(* IEC 61131-3 sources: teller/JD_Teller_LC2_V11/Class/TellerClass_Teller, 1 file *)

(* ---- TellerClass_Teller.st ---- *)
(*!
<Class
	Name               = "TellerClass_Teller"
	Revision           = "1.3"
	RealtimeTask       = "true"
	DefRealtime        = "1 ms"
	DefRealtimeIndex   = "1073742080"
	CyclicTask         = "true"
	DefCyclictime      = "100 ms"
	DefCyclicIndex     = "1073742080"
	BackgroundTask     = "true"
	DefBackground      = "200 ms"
	DefBackgroundIndex = "1073742080"
	Sigmatek           = "false"
	OSInterface        = "false"
	HighPriority       = "false"
	Automatic          = "false"
	UpdateMode         = "Prescan"
	SharedCommandTable = "true"
	Objectsize         = "(570,120)">
	<Channels>
		<Server Name="ClassSvr" Visualized="true" Initialize="false" WriteProtected="false" Retentive="false" Comment="Standaard 20&#13;&#10;"/>
		<Server Name="i2SenCNT" Visualized="true" Initialize="false" WriteProtected="false" Retentive="false" Comment="Servicemenu instelling&#13;&#10;&#13;&#10;Met de waarde kan het aantal telsensors worden ingesteld.&#13;&#10;Algemene instelling. Met deze server worden alle Visuteller &#13;&#10;i2SenCNT overschreven!&#13;&#10;&#13;&#10;Bereik&#13;&#10;&#13;&#10;0:&#13;&#10;Alleen SensorL wordt gebruikt bij type 1 t/m 5, behalve type 3.&#13;&#10;&#13;&#10;1:&#13;&#10;Zowel Sensor L en Sensor R worden gebruikt bij type 1t/m 5, behalve type 3.&#13;&#10;&#13;&#10;"/>
		<Server Name="iBoxlengthCNT" Visualized="true" Initialize="false" WriteProtected="false" Retentive="false"/>
		<Server Name="iBoxlengthCNT_Max" Visualized="true" Initialize="false" WriteProtected="true" Retentive="false"/>
		<Server Name="iBoxlengthCNT_Min" Visualized="true" Initialize="false" WriteProtected="true" Retentive="false"/>
		<Server Name="iBoxlengthJamL" Visualized="true" Initialize="false" WriteProtected="false" Retentive="false"/>
		<Server Name="iBoxlengthJamL_Max" Visualized="true" Initialize="false" WriteProtected="true" Retentive="false"/>
		<Server Name="iBoxlengthJamL_Min" Visualized="true" Initialize="false" WriteProtected="true" Retentive="false"/>
		<Server Name="iBoxlengthJamR" Visualized="true" Initialize="false" WriteProtected="false" Retentive="false"/>
		<Server Name="iBoxlengthJamR_Max" Visualized="true" Initialize="false" WriteProtected="true" Retentive="false"/>
		<Server Name="iBoxlengthJamR_Min" Visualized="true" Initialize="false" WriteProtected="true" Retentive="false"/>
		<Server Name="iBoxlengthJamSTR" Visualized="true" Initialize="false" WriteProtected="false" Retentive="false"/>
		<Server Name="iBoxlengthJamSTR_Max" Visualized="true" Initialize="false" WriteProtected="true" Retentive="false"/>
		<Server Name="iBoxlengthJamSTR_Min" Visualized="true" Initialize="false" WriteProtected="true" Retentive="false"/>
		<Server Name="iEncDiv" Visualized="true" Initialize="false" WriteProtected="false" Retentive="false" Comment="idem als iEncMul&#13;&#10;&#13;&#10;Alleen is dit de deelfactor"/>
		<Server Name="iEncMeetdist" Visualized="true" Initialize="false" WriteProtected="false" Retentive="false"/>
		<Server Name="iEncMul" Visualized="true" Initialize="false" WriteProtected="false" Retentive="false" Comment="Met deze instelling is de encoder in te stellen naar de juiste eenheid.&#13;&#10;&#13;&#10;Dit is de vermenigvuldig factor&#13;&#10;&#13;&#10; "/>
		<Server Name="iEncStapper" Visualized="true" Initialize="false" WriteProtected="false" Retentive="false"/>
		<Server Name="iJamdetReset" Visualized="true" Initialize="false" WriteProtected="false" Retentive="false"/>
		<Server Name="iSensorCNT" Visualized="true" Initialize="false" WriteProtected="false" Retentive="false" Comment="&#13;&#10;&#13;&#10;"/>
		<Server Name="iTotalProduction" Visualized="true" Initialize="false" WriteProtected="false" Retentive="false"/>
		<Server Name="MinSpot" Visualized="true" Initialize="false" WriteProtected="false" Retentive="false"/>
		<Server Name="oCounter" Visualized="true" Initialize="false" WriteProtected="false" Retentive="false"/>
		<Server Name="oCounterPerHour" Visualized="true" Initialize="false" WriteProtected="false" Retentive="false"/>
		<Server Name="oJamdetL" Visualized="true" Initialize="false" WriteProtected="true" Retentive="false"/>
		<Server Name="oJamdetR" Visualized="true" Initialize="false" WriteProtected="true" Retentive="false"/>
		<Server Name="oJamdetSTR" Visualized="true" Initialize="false" WriteProtected="true" Retentive="false"/>
		<Server Name="oRemainingProduction" Visualized="true" Initialize="false" WriteProtected="false" Retentive="false"/>
		<Server Name="oSensorHWCNT" Visualized="true" Initialize="false" WriteProtected="true" Retentive="false"/>
		<Server Name="oSpeed" Visualized="true" Initialize="false" WriteProtected="true" Retentive="false" Comment="Snelheid machine in m/min.&#13;&#10;&#13;&#10;in meter per minuut.&#13;&#10;"/>
		<Server Name="oStopperLSE" Visualized="true" Initialize="false" WriteProtected="false" Retentive="false" Comment="De serverLSE wordt gebruikt om plaatjes in LSE te laten zien"/>
		<Server Name="sAnalogSpeed_Man_Auto" Visualized="true" Initialize="false" WriteProtected="false" Retentive="false"/>
		<Server Name="sAnalogSpeedEnable" Visualized="true" Initialize="false" WriteProtected="false" Retentive="false"/>
		<Server Name="sCounter" Visualized="false" Initialize="false" WriteProtected="true" Retentive="false"/>
		<Server Name="sCounterPerMin" Visualized="false" Initialize="false" WriteProtected="true" Retentive="false"/>
		<Server Name="sData" Visualized="false" Initialize="false" WriteProtected="false" Retentive="SRam"/>
		<Server Name="SExtraBox" Visualized="true" Initialize="false" WriteProtected="false" Retentive="false" Comment="Standaard 30"/>
		<Server Name="sFactorAnalogSpeedIn" Visualized="true" Initialize="false" WriteProtected="false" Retentive="false" Comment="Slider voor bepaling van een factor voor aansturing van de conveyor met een analoog signaal&#13;&#10;&#13;&#10;Min = 0&#13;&#10;Max = 10000"/>
		<Server Name="sFactorAnalogSpeedout" Visualized="true" Initialize="false" WriteProtected="true" Retentive="false" Comment="&#13;&#10;Output voor snelheids referentie van de conveyor&#13;&#10;Factor voor aansturing van de conveyor met een analoog signaal&#13;&#10;&#13;&#10;Min = 0&#13;&#10;Max = 10000"/>
		<Server Name="SimSpeed" Visualized="true" Initialize="false" WriteProtected="false" Retentive="false"/>
		<Server Name="Simulatie" Visualized="true" Initialize="false" WriteProtected="false" Retentive="false"/>
		<Server Name="sMaxSpeed" Visualized="true" Initialize="false" WriteProtected="false" Retentive="false"/>
		<Server Name="sRemainingProduction" Visualized="false" Initialize="false" WriteProtected="true" Retentive="false"/>
		<Server Name="sTotalProduction" Visualized="false" Initialize="false" WriteProtected="true" Retentive="false"/>
		<Client Name="c_JamData" Required="true" Internal="false"/>
		<Client Name="cAnalogSpeedOut" Required="true" Internal="false"/>
		<Client Name="cExtBoxCount" Required="true" Internal="false"/>
		<Client Name="coCounter" Required="true" Internal="false"/>
		<Client Name="coCounterPerMin" Required="true" Internal="false"/>
		<Client Name="coRemainingproduction" Required="true" Internal="false"/>
		<Client Name="coSpeed" Required="true" Internal="false"/>
		<Client Name="coTotalproduction" Required="true" Internal="false"/>
		<Client Name="GetDataTanabe" Required="false" Internal="false"/>
		<Client Name="iEncoder" Required="false" Internal="false"/>
		<Client Name="iSensorL" Required="false" Internal="false"/>
		<Client Name="iSensorR" Required="false" Internal="false"/>
		<Client Name="iSensorSTR" Required="false" Internal="false"/>
		<Client Name="iSimPuls" Required="false" Internal="false"/>
		<Client Name="ObjTaskObjectControl" Required="false" Internal="false"/>
		<Client Name="oHeadnr01" Required="false" Internal="false"/>
		<Client Name="oHeadnr02" Required="false" Internal="false"/>
		<Client Name="oHeadnr03" Required="false" Internal="false"/>
		<Client Name="oHeadnr04" Required="false" Internal="false"/>
		<Client Name="oHeadnr05" Required="false" Internal="false"/>
		<Client Name="oHeadnr06" Required="false" Internal="false"/>
		<Client Name="oHeadnr07" Required="false" Internal="false"/>
		<Client Name="oHeadnr08" Required="false" Internal="false"/>
		<Client Name="oJam" Required="false" Internal="false"/>
		<Client Name="RamEx" Required="true" Internal="false"/>
		<Client Name="ri2SenCNT" Required="true" Internal="true"/>
		<Client Name="riBoxlengthCNT" Required="true" Internal="true"/>
		<Client Name="riBoxlengthJAML" Required="true" Internal="true"/>
		<Client Name="riBoxlengthJAMR" Required="true" Internal="true"/>
		<Client Name="riBoxlengthJamSTR" Required="true" Internal="true"/>
		<Client Name="riEncDiv" Required="true" Internal="true"/>
		<Client Name="riEncMul" Required="true" Internal="true"/>
		<Client Name="riSensorCNT" Required="true" Internal="true"/>
		<Client Name="riTotalProduction" Required="true" Internal="true"/>
		<Client Name="RMinSpot" Required="true" Internal="true"/>
		<Client Name="roCounter" Required="true" Internal="true"/>
		<Client Name="rsAnalogSpeedEnable" Required="true" Internal="true"/>
		<Client Name="rSextraBox" Required="true" Internal="true"/>
		<Client Name="rsFactorAnalogSpeedIn" Required="true" Internal="true"/>
		<Client Name="rsMaxSpeed" Required="true" Internal="true"/>
	</Channels>
	<RevDoku>
		<Owner Company="JD" Author="AP"/>
		<Dokumentation Revision="1.3" Date="2018-01-12" Author="AP" Company="JD" Description="Toevoegen extra counter output (cExBoxCount - CIO07) voor triggeren bij detectie van nieuwe doos&#13;&#10;"/>
		<Dokumentation Revision="1.2" Date="2016-10-24" Author="AP" Company="JD" Description="Aansturing Conveyor analoog signaal&#13;&#10;"/>
		<Dokumentation Revision="1.1" Date="2014-10-14" Author="SV" Company="JD" Description="ClassSvr teruggezet en server MinSpot opnieuw aangemaakt.&#13;&#10;coTotalproduction naar server Stotalproduction overzetten.&#13;&#10;coCounter naar server sCounter overzetten.&#13;&#10;coRemainingProduction naar server sRemainingProduction overzetten.&#13;&#10;coCounterPerMin naar server sCounterPerMin overzetten."/>
		<Dokumentation Revision="1.1" Date="2014-09-23" Author="SV" Company="JD" Description="TaskOnOff code uit class verwijderd. TaskOnOff server verwijderd."/>
		<Dokumentation Revision="1.0" Date="2014-09-04" Author="SV" Company="JD" Description="Gekopieert uit retrofit van versie 1.9. TellerClass_Teller geeft nu de waarden van EncMul, EncDiv,&#13;&#10;MinSpot en ExtraBox door aan de TeachInClass_Teller. Via de nieuwe client c_JamData.&#13;&#10;"/>
	</RevDoku>
	<Network Name="TellerClass_Teller">
		<!-- List of Components in this network -->
		<Components>
			<Object
				Name       = "ri2SenCNT"
				Class      = "Ram"
				Position   = "(210,1740)"
				Visualized = "true">
				<Channels>
					<Server Name="Data"/>
				</Channels>
			</Object>
			<Object
				Name       = "riBoxlengthCNT"
				Class      = "Ram"
				Position   = "(210,840)"
				Visualized = "true">
				<Channels>
					<Server Name="Data"/>
				</Channels>
			</Object>
			<Object
				Name       = "riBoxlengthJAML"
				Class      = "Ram"
				Position   = "(210,1290)"
				Visualized = "true">
				<Channels>
					<Server Name="Data"/>
				</Channels>
			</Object>
			<Object
				Name       = "riBoxlengthJAMR"
				Class      = "Ram"
				Position   = "(210,1440)"
				Visualized = "true">
				<Channels>
					<Server Name="Data"/>
				</Channels>
			</Object>
			<Object
				Name       = "riBoxlengthJamSTR"
				Class      = "Ram"
				Position   = "(210,1590)"
				Visualized = "true">
				<Channels>
					<Server Name="Data"/>
				</Channels>
			</Object>
			<Object
				Name       = "riEncDiv"
				Class      = "Ram"
				Position   = "(210,540)"
				Visualized = "true">
				<Channels>
					<Server Name="Data"/>
				</Channels>
			</Object>
			<Object
				Name       = "riEncMul"
				Class      = "Ram"
				Position   = "(210,390)"
				Visualized = "true">
				<Channels>
					<Server Name="Data"/>
				</Channels>
			</Object>
			<Object
				Name       = "riSensorCNT"
				Class      = "Ram"
				Position   = "(210,690)"
				Visualized = "true">
				<Channels>
					<Server Name="Data"/>
				</Channels>
			</Object>
			<Object
				Name       = "riTotalProduction"
				Class      = "Ram"
				Position   = "(210,990)"
				Visualized = "true">
				<Channels>
					<Server Name="Data"/>
				</Channels>
			</Object>
			<Object
				Name       = "RMinSpot"
				Class      = "Ram"
				Position   = "(210,90)"
				Visualized = "true">
				<Channels>
					<Server Name="Data"/>
				</Channels>
			</Object>
			<Object
				Name       = "roCounter"
				Class      = "Ram"
				Position   = "(210,1140)"
				Visualized = "true">
				<Channels>
					<Server Name="Data"/>
				</Channels>
			</Object>
			<Object
				Name       = "rsAnalogSpeedEnable"
				Class      = "Ram"
				Position   = "(210,2190)"
				Visualized = "true">
				<Channels>
					<Server Name="Data"/>
				</Channels>
			</Object>
			<Object
				Name       = "rSextraBox"
				Class      = "Ram"
				Position   = "(210,240)"
				Visualized = "true">
				<Channels>
					<Server Name="Data"/>
				</Channels>
			</Object>
			<Object
				Name       = "rsFactorAnalogSpeedIn"
				Class      = "Ram"
				Position   = "(210,2040)"
				Visualized = "true">
				<Channels>
					<Server Name="Data"/>
				</Channels>
			</Object>
			<Object
				Name       = "rsMaxSpeed"
				Class      = "Ram"
				Position   = "(210,1890)"
				Visualized = "true">
				<Channels>
					<Server Name="Data"/>
				</Channels>
			</Object>
		</Components>
		<Comments>
		</Comments>
		<!-- List of Connections in this network -->
		<Connections>
			<Connection Source="this.riTotalProduction" Destination="riTotalProduction.Data"/>
			<Connection Source="this.RMinSpot" Destination="RMinSpot.Data"/>
			<Connection Source="this.rSextraBox" Destination="rSextraBox.Data"/>
			<Connection Source="this.riEncMul" Destination="riEncMul.Data"/>
			<Connection Source="this.riEncDiv" Destination="riEncDiv.Data"/>
			<Connection Source="this.riSensorCNT" Destination="riSensorCNT.Data"/>
			<Connection Source="this.riBoxlengthCNT" Destination="riBoxlengthCNT.Data"/>
			<Connection Source="this.ri2SenCNT" Destination="ri2SenCNT.Data"/>
			<Connection Source="this.riBoxlengthJAML" Destination="riBoxlengthJAML.Data"/>
			<Connection Source="this.riBoxlengthJAMR" Destination="riBoxlengthJAMR.Data"/>
			<Connection Source="this.riBoxlengthJamSTR" Destination="riBoxlengthJamSTR.Data"/>
			<Connection Source="this.roCounter" Destination="roCounter.Data"/>
			<Connection Source="this.rsMaxSpeed" Destination="rsMaxSpeed.Data"/>
			<Connection Source="this.rsFactorAnalogSpeedIn" Destination="rsFactorAnalogSpeedIn.Data"/>
			<Connection Source="this.rsAnalogSpeedEnable" Destination="rsAnalogSpeedEnable.Data"/>
		</Connections>
		<!-- Headerfiles -->
		<Options>
		</Options>
	</Network>
</Class>
*)
TellerClass_Teller : CLASS
  //Servers:
	ClassSvr 	: SvrChCmd_DINT;
	MinSpot 	: SvrCh_DINT;
	SimSpeed 	: SvrCh_DINT;
	Simulatie 	: SvrCh_DINT;
	SExtraBox 	: SvrCh_DINT;
	iEncMul 	: SvrCh_DINT;
	iEncDiv 	: SvrCh_DINT;
	sMaxSpeed 	: SvrCh_DINT;
	iEncStapper 	: SvrCh_DINT;
	iEncMeetdist 	: SvrCh_DINT;
	oSpeed 	: SvrCh_DINT;
	iSensorCNT 	: SvrCh_DINT;
	oSensorHWCNT 	: SvrCh_DINT;
	iBoxlengthCNT 	: SvrCh_DINT;
	iTotalProduction 	: SvrCh_DINT;
	oRemainingProduction 	: SvrCh_DINT;
	oCounter 	: SvrCh_DINT;
	sAnalogSpeed_Man_Auto 	: SvrCh_DINT;
	sAnalogSpeedEnable 	: SvrCh_DINT;
	sFactorAnalogSpeedIn 	: SvrCh_DINT;
	sFactorAnalogSpeedout 	: SvrCh_DINT;
	oCounterPerHour 	: SvrCh_DINT;
	iBoxlengthJamL 	: SvrCh_DINT;
	iBoxlengthJamR 	: SvrCh_DINT;
	iBoxlengthJamSTR 	: SvrCh_DINT;
	oJamdetL 	: SvrCh_DINT;
	oJamdetR 	: SvrCh_DINT;
	oJamdetSTR 	: SvrCh_DINT;
	iJamdetReset 	: SvrCh_DINT;
	oStopperLSE 	: SvrCh_DINT;
	sData 	: SvrCh_DINT;
	i2SenCNT 	: SvrCh_DINT;
	iBoxlengthCNT_Max 	: SvrCh_DINT;
	iBoxlengthCNT_Min 	: SvrCh_DINT;
	iBoxlengthJamL_Max 	: SvrCh_DINT;
	iBoxlengthJamL_Min 	: SvrCh_DINT;
	iBoxlengthJamR_Max 	: SvrCh_DINT;
	iBoxlengthJamR_Min 	: SvrCh_DINT;
	iBoxlengthJamSTR_Max 	: SvrCh_DINT;
	iBoxlengthJamSTR_Min 	: SvrCh_DINT;
	sTotalProduction 	: SvrCh_DINT;
	sCounter 	: SvrCh_DINT;
	sRemainingProduction 	: SvrCh_DINT;
	sCounterPerMin 	: SvrCh_DINT;
  //Clients:
	iEncoder 	: CltCh_DINT;
	iSensorL 	: CltCh_DINT;
	iSensorR 	: CltCh_DINT;
	iSensorSTR 	: CltCh_DINT;
	oJam 	: CltCh_DINT;
	oHeadnr01 	: CltCh_DINT;
	oHeadnr02 	: CltCh_DINT;
	oHeadnr03 	: CltCh_DINT;
	oHeadnr04 	: CltCh_DINT;
	oHeadnr05 	: CltCh_DINT;
	oHeadnr06 	: CltCh_DINT;
	oHeadnr07 	: CltCh_DINT;
	oHeadnr08 	: CltCh_DINT;
	RamEx 	: CltChCmd_RAMex;
	RMinSpot 	: CltChCmd_Ram;
	rSextraBox 	: CltChCmd_Ram;
	riEncMul 	: CltChCmd_Ram;
	riEncDiv 	: CltChCmd_Ram;
	riSensorCNT 	: CltChCmd_Ram;
	riBoxlengthCNT 	: CltChCmd_Ram;
	riTotalProduction 	: CltChCmd_Ram;
	riBoxlengthJAML 	: CltChCmd_Ram;
	riBoxlengthJAMR 	: CltChCmd_Ram;
	riBoxlengthJamSTR 	: CltChCmd_Ram;
	roCounter 	: CltChCmd_Ram;
	ri2SenCNT 	: CltChCmd_Ram;
	iSimPuls 	: CltCh_DINT;
	coTotalproduction 	: CltCh_DINT;
	coCounter 	: CltCh_DINT;
	coRemainingproduction 	: CltCh_DINT;
	coCounterPerMin 	: CltCh_DINT;
	coSpeed 	: CltCh_DINT;
	c_JamData 	: CltChCmd_RAMex;
	GetDataTanabe 	: CltCh_DINT;
	rsMaxSpeed 	: CltChCmd_Ram;
	rsFactorAnalogSpeedIn 	: CltChCmd_Ram;
	cAnalogSpeedOut 	: CltCh_DINT;
	rsAnalogSpeedEnable 	: CltChCmd_Ram;
	ObjTaskObjectControl 	: CltChCmd__TaskObjectControl;
	cExtBoxCount 	: CltCh_DINT;
  //Variables:
		Sensor 	: SensorLR;
		Jam 	: Jam;
		Kop 	: Aansturing;
		Sposbuffer : ARRAY [0..10] OF ringbuffer;

		Enc 	: Encoder1;
		Kopdata 	: ^tKop;
		Teller 	: Counter1;
		Ospeedie 	: tOspeed;
		timer 	: UDINT;
		CounterperMinute 	: DINT;
		i 	: DINT;
		ii 	: DINT;
		MarkAktieInterupt : ARRAY [0..10] OF SINT;

		JamData 	: ^tJamDetect;
		tmp_AutoAnalogSpeed 	: DINT;
		tmp_ManualAnalogSpeed 	: DINT;
		MyobjInfo 	: LSLOBJ_INFO;
  //Functions:

	FUNCTION VIRTUAL GLOBAL Init;

	FUNCTION VIRTUAL GLOBAL CyWork
		VAR_INPUT
			EAX 	: UDINT;
		END_VAR
		VAR_OUTPUT
			state (EAX) 	: UDINT;
		END_VAR;

	FUNCTION VIRTUAL GLOBAL RtWork
		VAR_INPUT
			EAX 	: UDINT;
		END_VAR
		VAR_OUTPUT
			state (EAX) 	: UDINT;
		END_VAR;

	FUNCTION VIRTUAL GLOBAL Background
		VAR_INPUT
			EAX 	: UDINT;
		END_VAR
		VAR_OUTPUT
			state (EAX) 	: UDINT;
		END_VAR;

	FUNCTION GLOBAL GetSensorSprayer
		VAR_OUTPUT
			Result 	: DINT;
		END_VAR;

	FUNCTION GLOBAL GetSensorKicker
		VAR_OUTPUT
			Result 	: DINT;
		END_VAR;

	FUNCTION GLOBAL GetSensorOffsetSprayer
		VAR_OUTPUT
			Result 	: DINT;
		END_VAR;

	FUNCTION GLOBAL GetSensorOffsetKicker
		VAR_OUTPUT
			Result 	: DINT;
		END_VAR;

	FUNCTION GLOBAL SetMarkInterupt
		VAR_INPUT
			Sprayer_Kicker 	: DINT;			//! <Variable Comment="1 = sprayer&#13;&#10;2 = kicker" Name="SetMarkInterupt.Sprayer_Kicker"/>
		END_VAR;

	FUNCTION VIRTUAL GLOBAL sMaxSpeed::Write
		VAR_INPUT
			input (EAX) 	: DINT;
		END_VAR
		VAR_OUTPUT
			result (EAX) 	: DINT;
		END_VAR;

	FUNCTION VIRTUAL GLOBAL sAnalogSpeed_Man_Auto::Write
		VAR_INPUT
			input (EAX) 	: DINT;
		END_VAR
		VAR_OUTPUT
			result (EAX) 	: DINT;
		END_VAR;

	FUNCTION VIRTUAL GLOBAL sAnalogSpeedEnable::Write
		VAR_INPUT
			input (EAX) 	: DINT;
		END_VAR
		VAR_OUTPUT
			result (EAX) 	: DINT;
		END_VAR;

	FUNCTION VIRTUAL GLOBAL sFactorAnalogSpeedIn::Write
		VAR_INPUT
			input (EAX) 	: DINT;
		END_VAR
		VAR_OUTPUT
			result (EAX) 	: DINT;
		END_VAR;

	FUNCTION VIRTUAL GLOBAL sData::Read
		VAR_OUTPUT
			output (EAX) 	: DINT;
		END_VAR;
  //Tables:
	FUNCTION @STD
		VAR_OUTPUT
			ret_code	: CONFSTATES;
		END_VAR;
	FUNCTION GLOBAL TAB @CT_;
END_CLASS;

#pragma using Ram
#pragma usingLtd _TaskObjectControl
#pragma usingLtd RAMex

FUNCTION VIRTUAL GLOBAL TellerClass_Teller::Init

  if  RamEx.GetSize() <> sizeof(tKop) then
      RamEx.SetSize(udSize:=sizeof(tKop));
  end_if;

   //SV 29-08-2014
  if      c_JamData.GetSize() <> sizeof(tJamDetect) then
          c_JamData.SetSize(udSize:=sizeof(tJamDetect));
  end_if;

  if  _FirstScan = 1 then
      Kopdata := (RamEx.GetDataPtr())$^tKop;
      JamData := (c_JamData.GetDataPtr())$^tJamDetect;//SV
      //divider mag niet 0 zijn
      if iEncDiv = 0 then
         iEncDiv :=1;
      end_if;

      //geheugen uitlezen
      RMinSpot := RMinSpot.Read();
      MinSpot.Write(RMinSpot);
      rSExtraBox := rSExtraBox.Read();
      SextraBox.Write(rSExtraBox);
      riEncMul := riEncMul.Read();
      iEncMul.Write(riEncMul);
      riEncDiv := riEncDiv.Read();
      iEncDiv.Write(riEncDiv);
      riSensorCNT := riSensorCNT.Read();
      iSensorCNT.Write(riSensorCNT);
      riBoxlengthCNT := riBoxlengthCNT.Read();
      iBoxlengthCNT.Write(riBoxlengthCNT);
      riTotalProduction := riTotalProduction.Read();
      iTotalProduction.Write(riTotalProduction);
      rocounter := rocounter.Read();
      ocounter.Write(rocounter);
      riBoxlengthJAML := riBoxlengthJAML.Read();
      iBoxlengthJamL.Write(riBoxlengthJAML);
      riBoxlengthJAMR := riBoxlengthJAMr.Read();
      iBoxlengthJamr.Write(riBoxlengthJAMr);
      riBoxlengthJamSTR := riBoxlengthJAMstr.Read();
      iBoxlengthJamSTR.Write(riBoxlengthJamSTR);
      ri2SenCNT := ri2SenCNT.Read();
      i2SenCNT.Write(ri2SenCNT);
      rsFactorAnalogSpeedIn := rsFactorAnalogSpeedIn.Read();
      sFactorAnalogSpeedIn.Write(input:=rsFactorAnalogSpeedIn);
      rsMaxSpeed := rsMaxSpeed.Read();
      sMaxSpeed.Write(input:=rsMaxSpeed);
      rsAnalogSpeedEnable := rsAnalogSpeedEnable.Read();
      sAnalogSpeedEnable.Write(input:=rsAnalogSpeedEnable);

    //Verhouding Cyclustijd EncoderClass *50ms* en TellerClass *1ms*
      Enc.EncPerCycle := 50;

    //Encoder resolutie
      Enc.EncResolutie := 1000;

    //aantal dozen per uur
      teller.SpeedCalc:=0;
      oCounterPerHour:=0;
      iBoxlengthCNT_Max:=2000;
      iBoxlengthCNT_Min:=0;
      iBoxlengthJamL_Max:=2000;
      iBoxlengthJamL_Min:=0;
      iBoxlengthJamR_Max:=2000;
      iBoxlengthJamR_Min:=0;
      iBoxlengthJamSTR_Max:=2000;
      iBoxlengthJamSTR_Min:=0;

      ObjTaskObjectControl.GetObjectInfo(thispointer:=this, tasktype:=OBJ_CT, objinfo:=#MyobjInfo);

  end_if;

END_FUNCTION

FUNCTION VIRTUAL GLOBAL TellerClass_Teller::Background
	VAR_INPUT
		EAX 	: UDINT;
	END_VAR
	VAR_OUTPUT
		state (EAX) 	: UDINT;
	END_VAR

  //SV 14-10-2014 Client gegevens naar server zetten, tbv uitlezen serial tanabe class
  sTotalProduction := coTotalproduction;
  sCounter := coCounter;
  sRemainingProduction := coRemainingproduction;
  sCounterPerMin := coCounterPerMin;

      //Servers in Ram opslaan
        MinSpot := MinSpot.Read();
        RMinSpot.Write(MinSpot);
        SExtraBox := SExtraBox.Read();
        rSextraBox.Write(SExtraBox);
        iEncMul := iEncMul.Read();
        riEncMul.Write(iEncmul);
        iEncDiv := iEncDiv.Read();
        riEncDiv.Write(iEncDiv);
        iSensorCNT := iSensorCNT.Read();
        riSensorCNT.Write(iSensorCNT);
        iBoxlengthCNT := iBoxlengthCNT.Read();
        riBoxlengthCNT.Write(iBoxlengthCNT);
        iTotalProduction := iTotalProduction.Read();
        riTotalProduction.Write(iTotalProduction);
        iBoxlengthJamL := iBoxlengthJamL.Read();
        riBoxlengthJAML.Write(iBoxlengthJamL);
        iBoxlengthJamR := iBoxlengthJamR.Read();
        riBoxlengthJAMR.Write(iBoxlengthJamR);
        iBoxlengthJamSTR := iBoxlengthJamSTR.Read();
        riBoxlengthJamSTR.Write(iBoxlengthJamSTR);
        i2SenCNT := i2SenCNT.Read();
        ri2SenCNT.Write(i2SenCNT);

  //Snipperbeveiliging
        Sensor.MinimaleSpot:=MinSpot;  //standaard is dit 20

  //Jam, extra lengte die bij de doos wordt opgeteld
        Jam.SExtraBox := SExtraBox;  //30

  //Kop aansturing, extra lengte die bij de doos wordt opgeteld
        kop.SExtraBox := SExtraBox; // standaard is dit 30

  //Jam
        Jam.Boxlength[1] := iBoxlengthJamL;
        Jam.Boxlength[2] := iBoxlengthJamR;
        Jam.Boxlength[3] := iBoxlengthJamSTR;

  //Counter
        if    iBoxlengthCNT < 50 then
              iBoxlengthCNT := 50;
              iBoxlengthCNT.Write(iBoxlengthCNT);
        elsif iBoxlengthCNT > 2000 then
              iBoxlengthCNT := 2000;
              iBoxlengthCNT.Write(iBoxlengthCNT);
        end_if;

  // De server i2SenCNT bepaalt of er 1 of 2 telsensors worden gebruikt
        if    i2SenCNT < 0 then
              i2SenCNT:=0;
        elsif i2SenCNT > 1 then
              i2SenCNT:=1;
        end_if;

  //Aansturing van de koppen/Inlezen van Servers

      for kop.ii := 1 to kop.iii do

              //Mask van elke kop is gelijk aan mask van teller

                Kopdata^.Boxlengte[kop.ii] := iBoxlengthCNT;

              //welke fotocel

                if    Kopdata^.Sensor[kop.ii] = 1 then
                      Kop.Offset[kop.ii] := Kopdata^.OffsetL[Kop.ii];

                elsif Kopdata^.Sensor[kop.ii] = 2 then
                      Kop.Offset[kop.ii] := Kopdata^.OffsetR[Kop.ii];

                elsif Kopdata^.Sensor[kop.ii] = 3 then
                      Kop.Offset[kop.ii] := Kopdata^.OffsetSTR[Kop.ii];

                end_if;

              //Kopspecs inlezen
                Kop.Dooslengte[kop.ii] := (Kopdata^.Boxlengte[kop.ii] * Encres + Jam.SExtraBox * encres);

                Kop.StotAan[kop.ii] := (Kop.Offset[kop.ii] - Sensor.MinimaleSpot + Kopdata^.Start[kop.ii]); //afstand van sensor tot start spoor
                Kop.StotAan[kop.ii] := (Kop.StotAan[kop.ii] * Encres);

                Kop.StotUit[kop.ii] := (kop.Offset[kop.ii] - Sensor.MinimaleSpot + Kopdata^.Start[kop.ii] + Kopdata^.Lengte[kop.ii]); //afstand van sensor tot einde van spoor
                Kop.StotUit[kop.ii] := (Kop.StotUit[kop.ii] * Encres);

              //Met i2SenCNT wordt bepaald of er 1 of 2 telsensors aanwezig zijn
              //0->1 sensor, 1-> 2 sensoren
                if      i2SenCNT = 0 then
                        kopdata^.i2SensorCNT[kop.ii] := 0;
                        iSensorCNT := 1;

                elsif   i2SenCNT = 1 then
                        kopdata^.i2SensorCNT[kop.ii] := 1;
                        if iSensorCNT < 1 then
                           iSensorCNT := 1;
                        elsif iSensorCNT >2 then
                          iSensorCNT :=2;
                        end_if;
                end_if;

                Kopdata^.SensorHW[kop.ii]:= Sensor.DiHW[Kopdata^.Sensor[kop.ii]];
              //Pakket teller conveyor op 1 houden
                if  Kopdata^.iType[kop.ii] = 3 then
                    Kopdata^.Pakket1SET[kop.ii] := 1;
                    Kopdata^.Pakket2SET[kop.ii] := 0;
                end_if;

      end_for;

  // De server oStopperLSE wordt gebruikt als variabele om plaatjes in LSE te laten zien

      if      Kopdata^.iType[1] = 5 & Kopdata^.Present[1]| // Server "present"toegevoegd nadat de pulldown menus vervangen zijn door switch present (type blijft altijd gelijk)
              Kopdata^.iType[2] = 5 & Kopdata^.Present[2]|
              Kopdata^.iType[3] = 5 & Kopdata^.Present[3]|
              Kopdata^.iType[4] = 5 & Kopdata^.Present[4]|
              Kopdata^.iType[5] = 5 & Kopdata^.Present[5]|
              Kopdata^.iType[6] = 5 & Kopdata^.Present[6]|
              Kopdata^.iType[7] = 5 & Kopdata^.Present[7]|
              Kopdata^.iType[8] = 5 & Kopdata^.Present[8]then

              oStopperLSE := 1;
              oStopperLSE.Write(oStopperLSE);
      else
              oStopperLSE := 0;
              oStopperLSE.Write(oStopperLSE);

      end_if;

      Kopdata^.OutputHW[1]:= oHeadnr01;
      Kopdata^.OutputHW[2]:= oHeadnr02;
      Kopdata^.OutputHW[3]:= oHeadnr03;
      Kopdata^.OutputHW[4]:= oHeadnr04;
      Kopdata^.OutputHW[5]:= oHeadnr05;
      Kopdata^.OutputHW[6]:= oHeadnr06;
      Kopdata^.OutputHW[7]:= oHeadnr07;
      Kopdata^.OutputHW[8]:= oHeadnr08;

      Kop.iii  := 1;
      kop.iiii := 0;

      for ii:=1 to 8 do
         // De aantal keer dat for lussen in deze code wordt doorlopen
         if Kopdata^.iType[ii] > 0 then
            Kop.iii  := ii;
         end_if;

         //Bepaling hoevaak de for lus voor de sensoren en jamdetect worden doorlopen
         if Kopdata^.Sensor[ii] > kop.iiii then
            kop.iiii := Kopdata^.Sensor[ii];
         end_if;

      end_for;

      if  ops.tAbsolute - timer > 1000 then

          CounterperMinute        :=  oCounterPerHour;
          coTotalproduction       :=  iTotalProduction;
          coCounter               :=  oCounter;
          coRemainingproduction   :=  oRemainingProduction;
          coCounterPerMin         :=  to_dint(to_Real(CounterperMinute ) / 60);
          coSpeed                 :=  oSpeed;

          coTotalproduction.Write(input:=coTotalproduction);
          coCounter.Write(input:=coCounter);
          coRemainingproduction.Write(input:=coRemainingproduction);
          coCounterPerMin.Write(input:=coCounterPerMin);
          coSpeed.Write(input:=coSpeed);

          timer := ops.tAbsolute;

      end_if;

	state := READY;

END_FUNCTION

FUNCTION VIRTUAL GLOBAL TellerClass_Teller::CyWork
	VAR_INPUT
		EAX 	: UDINT;
	END_VAR
	VAR_OUTPUT
		state (EAX) 	: UDINT;
	END_VAR

    //encoder

      if iEncDiv = 0 then
         iEncDiv :=1;
      end_if;

      if    SimSpeed <= 0 then
            Enc.Multi   := iEncMul;
            Enc.Divider := iEncDiv;
      else

            Enc.Multi   := 1000;
            Enc.Divider := 60000;
      end_if;

      OSpeedie.EncIn :=iEncoder;
      ospeedie.EncDelta := OSpeedie.EncIn - OSpeedie.EncOud;
      OSpeedie.EncOud := OSpeedie.EncIn;
      oSpeed := to_dint((to_Real(ospeedie.EncDelta) * 60 * To_Real(Enc.Multi)) / (to_Real(Enc.Divider)*MyobjInfo.period));

      //Aansturing van de conveyor met een analoog signaal
      if    sAnalogSpeedEnable & sAnalogSpeed_Man_Auto=0 then //manual OFF
            if    tmp_AutoAnalogSpeed <> 0 then //oude waarde van sFactorAnalogSpeedIn weer activeren bij schakelen van manueel naar auto
                  tmp_ManualAnalogSpeed := sFactorAnalogSpeedIn;
                  sFactorAnalogSpeedIn := tmp_AutoAnalogSpeed;
                  tmp_AutoAnalogSpeed := 0;
            end_if;

            cAnalogSpeedOut := to_dint((to_real(oSpeed) * sFactorAnalogSpeedIn) / to_real(sMaxSpeed));

            if    cAnalogSpeedOut < 0 then
                  cAnalogSpeedOut := 0;
            elsif cAnalogSpeedOut > 10000 then
                  cAnalogSpeedOut := 10000;
            end_if;
      elsif sAnalogSpeedEnable & sAnalogSpeed_Man_Auto=1 then //manual ON
            if    tmp_AutoAnalogSpeed = 0 then //waarde van sFactorAnalogSpeedIn bewaren
                  tmp_AutoAnalogSpeed := sFactorAnalogSpeedIn;
            end_if;

            if    tmp_ManualAnalogSpeed > 0 then
                  sFactorAnalogSpeedIn := tmp_ManualAnalogSpeed;
                  tmp_ManualAnalogSpeed := 0;
            else
                  cAnalogSpeedOut := sFactorAnalogSpeedIn;
            end_if;
      else
            cAnalogSpeedOut := 0;
      end_if;

      if    sFactorAnalogSpeedout <> cAnalogSpeedOut then
            sFactorAnalogSpeedout := cAnalogSpeedOut;
            cAnalogSpeedOut.Write(input:=cAnalogSpeedOut);
      end_if;

    //De encoder multi wordt berekend (Dit nog testen)
          case  iEncStapper of

                  0:      //wachten todat lse de stapper ophoogd.
                          iEncMeetdist := 0;
                          iEncMeetdist.Write(iEncMeetdist);
                  1:
                          enc.Meting1 := iEncoder;    //startpositie van de encoder inlezen
                          enc.Meting2 := 0;
                          iEncStapper := 2;
                  2:                                  //LSE geeft opdracht de machineriem te verplaatsen

                  3:      enc.Meting2 :=  iEncoder;    //vervolgens wordt de stopposie van de encoder ingelezen
                          iEncStapper := 4;

                  4:
                          iEncMeetdist.Read();        //wachten totdat de afstand in mm wordt ingegeven

                          if   iEncMeetdist > 0  then

                          iEncDiv := 10000;
                          iEncDiv.Write(iEncDiv);     //De divider op 10000 zetten
                          riEncDiv.Write(input:=iEncDiv);

                          enc.encdiv := iEncDiv;
                          enc.enccalc1:= ENC.Meting2 - enc.Meting1;
                          enc.enccalc2:= enc.enccalc1 * enc.encdiv;
                          enc.enccalc3:= enc.enccalc2 / (iEncMeetdist*100);

                          iEncMul := enc.enccalc3;
                          iEncMul.Write(iEncMul);     //berekenen van de encoder multiplyer.
                          riEncMul.Write(input:=iEncMul);

                          iEncStapper := 0;
                          end_if;
          end_case;

    //Jam detect

         if    Jam.JamDetection[1] or Jam.JamDetection [2]  or Jam.JamDetection [3] then     //Bij Jamdetect L/R -> Client OJam hoog maken
               if   oJam = 0 then
                    oJam := 1;
                    oJam.Write(input:=Ojam);
               end_if;
         elsif oJam = 1 then
               oJam := 0;
               oJam.Write(input:=Ojam);
         end_if;

    //Counter1

         //welke telsensor
         if    iSensorCNT = 1  then
               oSensorHWCNT := iSensorL;
               oSensorHWCNT.Write(oSensorHWCNT);
         elsif iSensorCNT = 2  then
               oSensorHWCNT := iSensorR;
               oSensorHWCNT.Write(oSensorHWCNT);
         end_if;

         //Productie teller
         oRemainingProduction := iTotalProduction - oCounter;
         if oRemainingProduction < 0 then
            oRemainingProduction :=0;
         end_if;
         oRemainingProduction.Write(oRemainingProduction);

         //Teller Per uur
         if    oSpeed = 0 | ops.tAbsolute - Teller.Timer1 > 3000 then   //bij geen dozen of bij machine stilstand, na 3 seconden counter per uur op 0 zetten
               oCounterPerHour := 0;
               teller.wijzer:=0;
               teller.CaseNogTeProd:=0;
               Teller.SpeedCalc :=0;
         end_if;

         if    teller.Dist2Boxen = 0 then    //mag niet nul zijn!
               teller.Dist2Boxen:=1;
         end_if;

         if    teller.SpeedCalc & oSpeed > 0 then   //Hier krijgt de oCounterPerUur een waarde

               case teller.CaseNogTeProd of

               0:

                  teller.NogTeProdBuffer[teller.wijzer]:= ((oSpeed * 60 * 1000) / teller.Dist2Boxen);
                  teller.Timer := ops.tAbsolute;
                  teller.CaseNogTeProd:=1;

               1:

                  if ops.tAbsolute - Teller.Timer > 1000 then //om de seconde een waarde

                      if Teller.wijzer = 5 then
                          oCounterPerHour := ((teller.NogTeProdBuffer[1]+teller.NogTeProdBuffer[2]+teller.NogTeProdBuffer[3]+teller.NogTeProdBuffer[4]+teller.NogTeProdBuffer[5]) / Teller.wijzer);
                          oCounterPerHour.Write(input:=oCounterPerHour);
                      end_if;

                  if teller.wijzer = 5 then  //wijzer = 5 weer naar 1
                     teller.wijzer :=0;
                  end_if;

                  teller.wijzer+=1;
                  teller.CaseNogTeProd:=0;
                  end_if;

               end_case;

        end_if;

        if    oSpeed = 0 |
              ops.tAbsolute - Teller.Timer1 > 3000 then   //bij geen dozen of bij machine stilstand, na 3 seconden counter per uur op 0 zetten

              oCounterPerHour := 0;
              teller.wijzer:=0;

              teller.CaseNogTeProd:=0;
              Teller.SpeedCalc :=0;
        end_if;

        //Correcties bepalen
        for i:=1 to kop.iii do

        Kop.ScorAan[i]:=(enc.SpeedDelta * Kopdata^.TopkomInMs[i]);
        Kop.ScorUit[i]:=(enc.SpeedDelta * Kopdata^.TafvalInMs[i]);

        end_for;

  //SV 29-8-2014. Instellinen in de Jamdetection_TaechIn dezelfde waarde moeten hebben, zodat dit maar 1 keer hoeft te worden ingegeven.
  JamData^.MinSpot := MinSpot;
  JamData^.sExtraBox := SExtraBox;
  JamData^.iEncMulti := iEncMul;
  JamData^.iEncDiv := iEncDiv;

	state := READY;

END_FUNCTION

FUNCTION VIRTUAL GLOBAL TellerClass_Teller::RtWork
	VAR_INPUT
		EAX 	: UDINT;
	END_VAR
	VAR_OUTPUT
		state (EAX) 	: UDINT;
	END_VAR

//Als in de machine setup de functie is geselelecteerd wordt de code uitgevoerd

      if    SimSpeed <= 0 then
            iEncoder := iEncoder.Read();
      else
            iEncoder += SimSpeed;
      end_if;

      if    enc.Divider < 1 then
            enc.Divider := 1;
      end_if;

      Enc.EncoderDelta := iEncoder - Enc.EncoderOld;
      Enc.EncoderOld := iEncoder;
      Enc.SpeedDelta := ((Enc.EncoderDelta * encres * enc.Multi) / enc.Divider);

    //inlezen van de sensors

    //inlezen van de sensors
    //one shot op de ingang

            for Sensor.i := 1 to kop.iiii do

              //inlezen van de sensors
              if    Simulatie = 1 then
                    iSimPuls := iSimPuls.Read();
                    Sensor.DiHW[1] := iSimPuls;
                    Sensor.DiHW[2] := iSimPuls;
                    Sensor.DiHW[3] := iSimPuls;
              else
                    if Sensor.i = 1 then
                       iSensorL := iSensorL.Read();
                       Sensor.DiHW[1] := iSensorL;
                    end_if;
                    if Sensor.i = 2 then
                       iSensorR := iSensorR.Read();
                       Sensor.DiHW[2] := iSensorR;
                    end_if;
                    if Sensor.i = 3 then
                       iSensorSTR := iSensorSTR.Read();
                       Sensor.DiHW[3] := iSensorSTR;
                    end_if;
              end_if;

              case Sensor.MinimaalSSW[Sensor.i] of

              0:
                if  Sensor.DiHW[Sensor.i] then
                    Sensor.MinimaleCounter[Sensor.i]:=0;
                    Sensor.Din[Sensor.i]:=0;
                    Sensor.MinimaalSSW[Sensor.i]+=1;
                end_if;

              1:

                    Sensor.MinimaleCounter[Sensor.i]+= Enc.SpeedDelta;

                if  Sensor.MinimaleCounter[Sensor.i] > Sensor.MinimaleSpot * Encres then
                    if  Sensor.DiHW[Sensor.i] = 1 then
                        Sensor.Din[Sensor.i]:=1;
                    end_if;
                    Sensor.MinimaalSSW[Sensor.i]+=1;
                end_if;

              2:

                    Sensor.Din[Sensor.i]:=0;
                if  Sensor.DiHW[Sensor.i] =0 then
                    Sensor.MinimaalSSW[Sensor.i]:=0;
                end_if;

              end_case;
            end_for;

    //Jam

            for Jam.i := 1 to kop.iiii do

                 if (jam.Boxlength[Jam.i] <> 0) then

                      case Jam.CaseJam[Jam.i] of

                      0: //controleren of aan de snipper beveiliging is voldaan
                         if Sensor.Din[Jam.i] then
                            Jam.CaseJam[Jam.i] += 1;
                            Jam.JamPos[Jam.i] := Sensor.MinimaleSpot * encres;
                            Jam.JamBoxlength[Jam.i] := (jam.Boxlength[Jam.i] + Jam.SExtraBox) * encres;
                         end_if;

                      1: //Controle op Jamdetect
                         //Kijken of de sensor hoog is na de ingestelde Boxlengte en extra waarde

                             Jam.JamPos[Jam.i] += Enc.SpeedDelta;
                             if   Jam.JamPos[Jam.i] > Jam.JamBoxlength[Jam.i] then
                                if  Sensor.DiHW[Jam.i] then
                                    Jam.JamDetection [Jam.i] := 1;
                                    oJamdetL := Jam.JamDetection[1];
                                    oJamdetL.Write(input:=oJamdetL);
                                    oJamdetR := Jam.JamDetection[2];
                                    oJamdetR.Write(input:=oJamdetR);
                                    oJamdetSTR := Jam.JamDetection[3];
                                    oJamdetSTR.Write(input:=oJamdetSTR);
                                    Jam.CaseJam[Jam.i] += 1;

                                else
                                    Jam.JamDetection[Jam.i] := 0;   //Geen Jamdetect, terug naar stap 0 en wachten op een nieuwe doos
                                    oJamdetL := Jam.JamDetection[1];
                                    oJamdetL.Write(input:=oJamdetL);
                                    oJamdetR := Jam.JamDetection[2];
                                    oJamdetR.Write(input:=oJamdetR);
                                    oJamdetSTR := Jam.JamDetection[3];
                                    oJamdetSTR.Write(input:=oJamdetSTR);
                                    Jam.CaseJam[Jam.i] := 0;
                                end_if;

                             end_if;

                      2:  //Jam, reset is nodig om verder te gaan.

                         if iJamdetReset then
                            Jam.JamDetection[Jam.i] := 0;
                            oJamdetL := Jam.JamDetection[1];
                            oJamdetL.Write(input:=oJamdetL);
                            oJamdetR := Jam.JamDetection[2];
                            oJamdetR.Write(input:=oJamdetR);
                            oJamdetSTR := Jam.JamDetection[3];
                            oJamdetSTR.Write(input:=oJamdetSTR);
                            Jam.CaseJam[Jam.i]:=0;

                         end_if;

                      end_case;

                 else

                 //Als bij een jamdetect de waarde 0 wordt ingevoerd wordt de jam case gereset
                        if  Jam.JamDetection[Jam.i]  then
                            Jam.CaseJam[Jam.i]:=0;
                            Jam.JamDetection[Jam.i] := 0;

                              if  jam.i = 1 then
                                  oJamdetL := Jam.JamDetection[1];
                                  oJamdetL.Write(input:=oJamdetL);
                              end_if;

                              if  jam.i = 2 then
                                  oJamdetR := Jam.JamDetection[2];
                                  oJamdetR.Write(input:=oJamdetR);
                              end_if;

                              if  jam.i = 3 then
                                  oJamdetSTR := Jam.JamDetection[3];
                                  oJamdetSTR.Write(input:=oJamdetSTR);
                              end_if;
                        end_if;
                 end_if;

           end_for;

    //Counter1

          case Teller.i of

          0:
             if (( iSensorCNT = 1 & Sensor.Din[1] ) | ( iSensorCNT = 2 & Sensor.Din[2] )) then
                Teller.i += 1;
                Teller.CounterPos := Sensor.MinimaleSpot * Encres;
                teller.CounterBoxlength :=(iBoxlengthCNT + Jam.SExtraBox - Sensor.MinimaleSpot) * ENCRES;

                //Externe teller
                cExtBoxCount := 1;
                cExtBoxCount.Write(input:=cExtBoxCount);
             end_if;

          1:
                 Teller.CounterPos += Enc.SpeedDelta;
                 if   Teller.CounterPos > Teller.CounterBoxlength then
                      oCounter += 1;
                      Teller.Timer1 := ops.tAbsolute;
                      roCounter.Write(oCounter);
                      Teller.i += 1;
                      Teller.Dist2Boxen := (((iEncoder - teller.EncoderOLD) * Enc.Multi) / Enc.Divider);  //in mm

                      //Externe teller
                      cExtBoxCount := 0;
                      cExtBoxCount.Write(input:=cExtBoxCount);
                 end_if;

          2:

               Teller.i := 0;
               Teller.EncoderOLD := iEncoder;
               Teller.TelCalc +=1;

               if Teller.TelCalc = 3 then
                  Teller.TelCalc :=0;
                  Teller.SpeedCalc := 1;

               end_if;
          end_case;

    //Aansturing koppen

          for Kop.i:= 1 to kop.iii do

          //Hier wordt de encoderpositie van de doos opgeslagen in een ringbuffer
            case kop.CaseRing[kop.i] of

            0:
              if sensor.din[Kopdata^.Sensor[kop.i]] then
                 kop.CaseRing[kop.i]+=1;
                 Kop.Senpos[kop.i]:= Sensor.MinimaleSpot * ENCRES;
                 kop.wrpoint[kop.i]:=kop.wrpoint[kop.i] and 16#0000000F;
                 SPosbuffer[kop.i][kop.wrpoint[kop.i]] := iEncoder;  //Positie van de doos = sensor + snipperbeveiliging
                 kop.wrpoint[kop.i]+=1;
                 kop.wrpoint[kop.i]:=kop.wrpoint[kop.i] and 16#0000000F;
              end_if;

            1:

              Kop.Senpos[kop.i] += enc.SpeedDelta;

              if  Kop.Senpos[kop.i] > kop.Dooslengte[kop.i] then  //als de dooslengte + 30mm gemeten is kan weer een nieuwe doos in het buffer worden opgeslagen
                  Kop.CaseRing[kop.i]:=0;
              end_if;

            end_case;

         //Hier wordt de kop aangestuurd
            case  Kop.CaseAansturing[kop.i] of

            0: //Hebben we een nieuwe doos?

              if kop.wrpoint[kop.i] <> kop.rdpoint[kop.i] Then
                 // go
                 kop.rdpoint[kop.i]:=kop.rdpoint[kop.i] and 16#0000000F;
                 //positie berekenen van de doos
                 kop.Spos[kop.i]:= ((iEncoder-Sposbuffer[Kop.i][kop.rdpoint[kop.i]])*((enc.Multi*Encres)/enc.Divider));
                 kop.rdpoint[kop.i]+=1;
                 kop.rdpoint[kop.i]:=kop.rdpoint[kop.i] and 16#0000000F;

                 //Koppen aan
                 if   (Kopdata^.OnOff[kop.i] & Kopdata^.Present[kop.i]) | MarkAktieInterupt[kop.i] = 1 then
                      Kop.CaseAansturing[kop.i]+=1;
                 end_if;
              End_if;

            1:  //Kop aan
                kop.Spos[kop.i]+=enc.SpeedDelta;

                if    (Kop.Spos[kop.i] >= (kop.StotAan[kop.i] - Kop.ScorAan[kop.i])) then

                       if   MarkAktieInterupt[kop.i] = 0 then

                            if      Kopdata^.Pakket2SET[kop.i] = 0 then
                                    Kop.PakketWijzer[kop.i] := 0;
                            end_if;

                            if      Kop.PakketWijzer[kop.i] = 0  then
                                    Kopdata^.Pakket1[kop.i]+=1;
                            elsif   Kop.PakketWijzer[kop.i] = 1  then
                                    Kopdata^.Pakket2[kop.i]+=1;
                            end_if;

                            if      Kopdata^.Pakket1[kop.i] > Kopdata^.Pakket1SET[kop.i] then
                                    Kopdata^.Pakket1[kop.i] := 1;
                            end_if;

                            //pakket teller 1
                            if      Kopdata^.Pakket1[kop.i] = Kopdata^.Pakket1SET[kop.i] & Kop.PakketWijzer[kop.i] = 0 then
                                    Kop.Out[kop.i]:=1;
                                    Kop.CaseAansturing[kop.i]+=1;
                                    Kopdata^.Pakket2[kop.i] :=0;
                                    if  Kopdata^.Pakket2SET[kop.i] = 0 then
                                        Kop.PakketWijzer[kop.i] := 0;
                                    else
                                        Kop.PakketWijzer[kop.i] := 1;
                                    end_if;
                            //pakket teller 2
                            elsif   Kopdata^.Pakket2[kop.i] = Kopdata^.Pakket2SET[kop.i] & Kop.PakketWijzer[kop.i] = 1 then
                                    Kop.Out[kop.i]:=1;
                                    Kop.CaseAansturing[kop.i]+=1;
                                    Kopdata^.Pakket1[kop.i] :=0;
                                    Kop.PakketWijzer[kop.i] := 0;
                            else
                                    Kop.CaseAansturing[kop.i]+=1;
                            end_if;
                       else
                            Kop.Out[kop.i]:=1;
                            Kop.CaseAansturing[kop.i]+=1;
                            MarkAktieInterupt[kop.i] := 0;
                       end_if;
                end_if;
            2:
                  //Conveyor spoor
                  if    (Kopdata^.iType[kop.i] = 3 & (Kopdata^.Lengte[kop.i] > Kopdata^.Boxlengte[kop.i])) then //bij conveyor aansturing en dat lengte groter is dan boxlengte naar stap 6 voor afhandeling.
                        Kop.conveyor[kop.i]:=1;
                        kop.ConveyorPosdoos[kop.i]:= kop.Spos[kop.i];
                        kop.UpdateConv[kop.i]:=1;

                        kop.CaseAansturing[kop.i] :=0;

                  elsif (Kopdata^.iType[kop.i] = 3 & (kopdata^.Lengte[kop.i] <= Kopdata^.Boxlengte[kop.i])) then
                        kop.conveyor[kop.i]:=0;
                        Kop.CaseAansturing[kop.i]+=1;
                  else
                        Kop.CaseAansturing[kop.i]+=1;
                  end_if;

            3:     //Kop uitschakelen
                  kop.Spos[kop.i]+=enc.SpeedDelta;
                  if Kop.Spos[kop.i]>= (Kop.StotUit[kop.i]-kop.ScorUit[kop.i]) then
                            Kop.out[kop.i]:=0;
                            Kop.CaseAansturing[kop.i]:=0;
                  end_if;

            end_case;

            //als de lengte van het spoor groter is dan de boxlengte (kan alleen bij type 3 conveyor)
            //dan is de lengte, de afstand tussen 2 dozen. Dit om de conveyor continu te laten draaien
            case  kop.ConveyorCase[kop.i] of

            0:
                  if  kop.conveyor[kop.i] then

                  kop.ConveyorCase[kop.i] +=1;
                  kop.UpdateConv[kop.i]:=0;
                  kop.ConveyorPosDoosNew[kop.i]:= kop.ConveyorPosdoos[kop.i] + (kopdata^.Lengte[kop.i] * encres);                   //(kop.ConveyorPosdoos[kop.i] + kopdata^.Lengte[kop.i] * encres);// mod 200000;
                  kop.ConveyorLoper[kop.i]:=kop.ConveyorPosdoos[kop.i];
                  end_if;

            1:
                  kop.ConveyorLoper[kop.i] += enc.SpeedDelta;

                  if   kop.ConveyorLoper[kop.i] > kop.ConveyorPosDoosNew[kop.i] then
                       kop.ConveyorCase[kop.i] +=1;

                  elsif Kop.UpdateConv[kop.i] = 1 then
                       kop.ConveyorCase[kop.i] :=0;

                  end_if;

            2: //uitschakelen conveyor
                  kop.out[kop.i] := 0;
                  Kop.ConveyorCase[kop.i] :=0;
                  kop.conveyor[kop.i]:=0;

              end_case;

            //Minimale snelheid force Out
            if  oSpeed < Kopdata^.MinSpeed[kop.i] then
                kop.out[kop.i] := 0;
            end_if;

    end_for;

    //aansturing van de hardware + Testknop

      //kop1
      if  kop.Out[1] | Kopdata^.Test[1] then
          oHeadnr01 := 1;
      else
          oHeadnr01 := 0;
      end_if;

      //kop2
      if  kop.Out[2] | Kopdata^.Test[2] then
          oHeadnr02 := 1;
      else
          oHeadnr02 := 0;
      end_if;

      //kop3
      if  kop.Out[3] | Kopdata^.Test[3] then
          oHeadnr03 := 1;
      else
          oHeadnr03 := 0;
      end_if;

      //kop4
      if  kop.Out[4] | Kopdata^.Test[4] then
          oHeadnr04 := 1;
      else
          oHeadnr04 := 0;
      end_if;

      //kop5
      if  kop.Out[5] | Kopdata^.Test[5] then
          oHeadnr05 := 1;
      else
          oHeadnr05 := 0;
      end_if;

      //kop6
      if  kop.Out[6] | Kopdata^.Test[6] then
          oHeadnr06 := 1;
      else
          oHeadnr06 := 0;
      end_if;

      //kop7
      if  kop.Out[7] | Kopdata^.Test[7] then
          oHeadnr07 := 1;
      else
          oHeadnr07 := 0;
      end_if;

      //kop8
      if  kop.Out[8] | Kopdata^.Test[8] then
          oHeadnr08 := 1;
      else
          oHeadnr08 := 0;
      end_if;

      oHeadnr01.Write(oHeadnr01);
      oHeadnr02.Write(oHeadnr02);
      oHeadnr03.Write(oHeadnr03);
      oHeadnr04.Write(oHeadnr04);
      oHeadnr05.Write(oHeadnr05);
      oHeadnr06.Write(oHeadnr06);
      oHeadnr07.Write(oHeadnr07);
      oHeadnr08.Write(oHeadnr08);

	state := READY;

END_FUNCTION

FUNCTION VIRTUAL GLOBAL TellerClass_Teller::sData::Read
	VAR_OUTPUT
		output (EAX) 	: DINT;
	END_VAR

  sData:=(#Kopdata^)$dint;

	output := sData;

END_FUNCTION

FUNCTION GLOBAL TellerClass_Teller::GetSensorSprayer
	VAR_OUTPUT
		Result 	: DINT;
	END_VAR

  Result := Sensor.DiHW[2];

END_FUNCTION

FUNCTION GLOBAL TellerClass_Teller::GetSensorKicker
	VAR_OUTPUT
		Result 	: DINT;
	END_VAR

  Result := Sensor.DiHW[1];

END_FUNCTION

FUNCTION GLOBAL TellerClass_Teller::GetSensorOffsetSprayer
	VAR_OUTPUT
		Result 	: DINT;
	END_VAR

  Result := Kop.Offset[2];

END_FUNCTION

FUNCTION GLOBAL TellerClass_Teller::GetSensorOffsetKicker
	VAR_OUTPUT
		Result 	: DINT;
	END_VAR

  Result := Kop.Offset[1];

END_FUNCTION

FUNCTION GLOBAL TellerClass_Teller::SetMarkInterupt
	VAR_INPUT
		Sprayer_Kicker 	: DINT;
	END_VAR

  if    Sprayer_Kicker = 1 then //sprayer
        MarkAktieInterupt[1] := 1;
  elsif Sprayer_Kicker = 2 then //kicker
        MarkAktieInterupt[2] := 1;
  end_if;

END_FUNCTION

FUNCTION VIRTUAL GLOBAL TellerClass_Teller::sMaxSpeed::Write
	VAR_INPUT
		input (EAX) 	: DINT;
	END_VAR
	VAR_OUTPUT
		result (EAX) 	: DINT;
	END_VAR

  if    input < 120 then
        sMaxSpeed := 120;
  elsif input > 500 then
        sMaxSpeed := 500;
  else
        sMaxSpeed := input;
  end_if;

  rsMaxSpeed.Write(input:=sMaxSpeed);

	result := sMaxSpeed;

END_FUNCTION

FUNCTION VIRTUAL GLOBAL TellerClass_Teller::sFactorAnalogSpeedIn::Write
	VAR_INPUT
		input (EAX) 	: DINT;
	END_VAR
	VAR_OUTPUT
		result (EAX) 	: DINT;
	END_VAR

  if    input < 0 then
        sFactorAnalogSpeedIn := 0;
  elsif input > 10000 then
        sFactorAnalogSpeedIn := 10000;
  else
        sFactorAnalogSpeedIn := input;
  end_if;

  rsFactorAnalogSpeedIn.Write(input:=sFactorAnalogSpeedIn);

	result := sFactorAnalogSpeedIn;

END_FUNCTION

FUNCTION VIRTUAL GLOBAL TellerClass_Teller::sAnalogSpeedEnable::Write
	VAR_INPUT
		input (EAX) 	: DINT;
	END_VAR
	VAR_OUTPUT
		result (EAX) 	: DINT;
	END_VAR

  if    input <> 1 then
        sAnalogSpeedEnable := 0;
  else
        sAnalogSpeedEnable := input;
  end_if;

  rsAnalogSpeedEnable.Write(input:=sAnalogSpeedEnable);

	result := sAnalogSpeedEnable;

END_FUNCTION

FUNCTION VIRTUAL GLOBAL TellerClass_Teller::sAnalogSpeed_Man_Auto::Write
	VAR_INPUT
		input (EAX) 	: DINT;
	END_VAR
	VAR_OUTPUT
		result (EAX) 	: DINT;
	END_VAR

	sAnalogSpeed_Man_Auto := input;
	result := sAnalogSpeed_Man_Auto;

END_FUNCTION
